_actorStartMovingTimeoutArray[_currentActorStartMovingTimeoutIndex].ActorStartMovingTimeout.register(stEventEntity, timerTime, conformation, waitHWConformation);
_actorStartMovingTimeoutArray[_currentActorStartMovingTimeoutIndex].actorID := actorID;
_actorStartMovingTimeoutArray[_currentActorStartMovingTimeoutIndex].actorPtr := actorPtr;
_actorStartMovingTimeoutArray[_currentActorStartMovingTimeoutIndex].expectedActorValue := expectedActorValue;
_actorStartMovingTimeoutArray[_currentActorStartMovingTimeoutIndex].sensorID := sensorID;
_actorStartMovingTimeoutArray[_currentActorStartMovingTimeoutIndex].sensorPtr := sensorPtr;

register := TRUE;
RETURN;
END_METHOD

// resets all ActorStartMovingTimeouts
METHOD resetAll : BOOL
VAR_INPUT
END_VAR

VAR
	i : UINT;
END_VAR
// reset all alarms
FOR i := 0 TO _currentActorStartMovingTimeoutIndex DO
	_actorStartMovingTimeoutArray[i].ActorStartMovingTimeout.reset();
END_FOR

resetAll := TRUE;
RETURN;
END_METHOD

METHOD PRIVATE resolveWatchdogInput : BOOL
VAR_INPUT
	ActorStartMovingTimeoutEx : ActorStartMovingtimeoutEx_t;
END_VAR

VAR
	_tmpStr : STRING;
	
	_sensorVal : BOOL := FALSE; 
	_actorVal : BOOL := FALSE;
END_VAR
IF _IOExpantionHandler = NULL AND _IOExpantionHandlerNotValidErrorSent = FALSE THEN
	_IOExpantionHandlerNotValidErrorSent := TRUE;
	_ErrorMessage.CreateEx(TC_EVENTS.ProgrammingErrors.NoValidPointerToIOExpantionHandler, 0 );
	_ErrorMessage.ipArguments.AddString(__POUNAME());
	_tmpStr := formatPosition(__POSITION());
	_ErrorMessage.ipArguments.AddString(_tmpStr);
	_ErrorMessage.Send(0);
	resolveWatchdogInput := FALSE;
	RETURN;
END_IF

// reslove sensor value
IF ActorStartMovingTimeoutEx.sensorPtr <> NULL THEN
	_sensorVal := ActorStartMovingTimeoutEx.sensorPtr^;
ELSIF ActorStartMovingTimeoutEx.sensorID <> sensorID_t.SENSOR_NO_SENSOR THEN
	_sensorVal := _IOExpantionHandler^.getSensorStatus(ActorStartMovingTimeoutEx.sensorID);
END_IF

// reslove actor value
IF ActorStartMovingTimeoutEx.actorPtr <> NULL THEN
	_actorVal := ActorStartMovingTimeoutEx.actorPtr^;
ELSIF ActorStartMovingTimeoutEx.actorID <> actorID_t.ACTOR_NO_ACTOR THEN
	_actorVal := _IOExpantionHandler^.getActor(ActorStartMovingTimeoutEx.actorID);
END_IF

IF _sensorVal = FALSE THEN // ignore cases when sensor isn't active
	resolveWatchdogInput := TRUE; 
	RETURN; 
END_IF

IF ActorStartMovingTimeoutEx.expectedActorValue <> _actorVal THEN
	resolveWatchdogInput := FALSE; // value missmatch, start timeout
	RETURN;
END_IF

resolveWatchdogInput := TRUE; 
RETURN;
END_METHOD

// sets the IOExpantionHandler refferance
METHOD setIOExpantionHandler : BOOL
VAR_INPUT
	IOExpantionHandlerPtr: POINTER TO IOExpantionHandler_t;
END_VAR
_IOExpantionHandler := IOExpantionHandlerPtr;
setIOExpantionHandler := TRUE;
RETURN;
END_METHOD

METHOD update : BOOL
VAR_INPUT
END_VAR

VAR
	i : UINT;
END_VAR
FOR i := 0 TO _currentActorStartMovingTimeoutIndex DO
	_actorStartMovingTimeoutArray[i].ActorStartMovingTimeout.update(resolveWatchdogInput(_actorStartMovingTimeoutArray[i]));
END_FOR

update := TRUE;
RETURN;
END_METHOD

END_FUNCTION_BLOCK

// ---- POUs/ErrorSystem/PrimitiveWatchdogManager_t.TcPOU
FUNCTION_BLOCK PrimitiveWatchdogManager_t
VAR_INPUT
END_VAR
VAR_OUTPUT
END_VAR
VAR
	_primitiveWatchdogArray : ARRAY [0..99] OF  PrimitiveWatchdogEx_t;
	_maxPrimitiveWatchdogIndex : UINT := 99;
	_currentPrimitiveWatchdogIndex : UINT := 0;
	_ErrorMessage : FB_TcMessage;
	_IOExpantionHandler : POINTER TO IOExpantionHandler_t := NULL;
	
	_IOExpantionHandlerNotValidErrorSent : BOOL := FALSE;
END_VAR

// clears and destroyes all PrimetiveWatchdogs
METHOD clear : BOOL
VAR_INPUT
END_VAR
_currentPrimitiveWatchdogIndex := 0;

clear := TRUE;
RETURN;
END_METHOD

// confirm all primitiveWatchdogs
METHOD confirmAll : BOOL
VAR_INPUT
END_VAR

VAR
	i: UINT;
END_VAR
// confirm all alarms
FOR i := 0 TO _currentPrimitiveWatchdogIndex DO
	_primitiveWatchdogArray[i].primitiveWatchdog.confirm();
END_FOR

confirmAll := TRUE;
RETURN;
END_METHOD

// if true an error has been trown
METHOD hasError : BOOL
VAR_INPUT
END_VAR

VAR
	i: UINT;
END_VAR
FOR i := 0 TO _currentPrimitiveWatchdogIndex DO
	hasError := hasError OR THIS^._primitiveWatchdogArray[i].primitiveWatchdog.isAlarmRaised();
END_FOR

RETURN;
END_METHOD

METHOD register : BOOL
VAR_INPUT
	stEventEntity : TcEventEntry;
	timerTime : TIME; // sets the timer for the timeout
	conformation : BOOL := TRUE;
	invert : BOOL := FALSE; // if true, inverts the watchdog feeding signal
	sensorID : sensorID_t := sensorID_t.SENSOR_NO_SENSOR;
	sensorPtr : POINTER TO BOOL := NULL;
	waitHWConformation : BOOL := TRUE;
END_VAR
VAR
	_tmpStr : STRING;
END_VAR
IF _currentPrimitiveWatchdogIndex + 1 > _maxPrimitiveWatchdogIndex THEN
	_ErrorMessage.CreateEx(TC_EVENTS.ProgrammingErrors.ExceedingAllowedAmountOfPrimitiveWatchdogTimeouts, 0 );
	_ErrorMessage.ipArguments.AddString(__POUNAME());
	_tmpStr := formatPosition(__POSITION());
	_ErrorMessage.ipArguments.AddString(_tmpStr);
	_ErrorMessage.ipArguments.AddUInt(_maxPrimitiveWatchdogIndex);
	_ErrorMessage.Send(0);
	
	register := FALSE;
	RETURN;
END_IF

IF (NOT(sensorID = sensorID_t.SENSOR_NO_SENSOR XOR sensorPtr = NULL)) THEN
	_ErrorMessage.CreateEx(TC_EVENTS.ProgrammingErrors.primitiveWatchdogNoValidSensorGiven, 0 );
	_ErrorMessage.ipArguments.AddString(__POUNAME());
	_tmpStr := formatPosition(__POSITION());
	_ErrorMessage.ipArguments.AddString(_tmpStr);
	_ErrorMessage.Send(0);
	
	register := FALSE;
	RETURN;
END_IF

_currentPrimitiveWatchdogIndex := _currentPrimitiveWatchdogIndex + 1; // increase it by one

_primitiveWatchdogArray[_currentPrimitiveWatchdogIndex].primitiveWatchdog.register(stEventEntity, timerTime, conformation, waitHWConformation);

_primitiveWatchdogArray[_currentPrimitiveWatchdogIndex].sensorID := sensorID;
_primitiveWatchdogArray[_currentPrimitiveWatchdogIndex].sensorPtr := sensorPtr;
_primitiveWatchdogArray[_currentPrimitiveWatchdogIndex].invert := invert;

register := TRUE;
RETURN;
END_METHOD

// resets all primitiveTimeouts
METHOD resetAll : BOOL
VAR_INPUT
END_VAR

VAR
	i: UINT;
END_VAR
// reset all alarms
FOR i := 0 TO _currentPrimitiveWatchdogIndex DO
	_primitiveWatchdogArray[i].primitiveWatchdog.reset();
END_FOR

resetAll := TRUE;
RETURN;
END_METHOD

METHOD PRIVATE resolveWatchdogImput : BOOL
VAR_INPUT
	PrimitiveWatchdogEx : PrimitiveWatchdogEx_t;
END_VAR

IF PrimitiveWatchdogEx.sensorID <> sensorID_t.SENSOR_NO_SENSOR THEN
	resolveWatchdogImput := _IOExpantionHandler^.getSensorStatus(PrimitiveWatchdogEx.sensorID);
END_IF

IF PrimitiveWatchdogEx.sensorPtr <> NULL THEN
	resolveWatchdogImput := PrimitiveWatchdogEx.sensorPtr^;
END_IF

IF PrimitiveWatchdogEx.invert THEN
	resolveWatchdogImput := NOT resolveWatchdogImput;
END_IF

RETURN;
END_METHOD

METHOD setIOExpantionHandler : BOOL
VAR_INPUT
	IOExpantionHandlerPtr: POINTER TO IOExpantionHandler_t;
END_VAR
_IOExpantionHandler := IOExpantionHandlerPtr;
setIOExpantionHandler := TRUE;
RETURN;
END_METHOD

METHOD update : BOOL
VAR_INPUT
END_VAR

VAR
	i: UINT;
END_VAR
FOR i := 0 TO _currentPrimitiveWatchdogIndex DO
	_primitiveWatchdogArray[i].primitiveWatchdog.update(resolveWatchdogImput(_primitiveWatchdogArray[i]));
END_FOR

update := TRUE;
RETURN;
END_METHOD

END_FUNCTION_BLOCK

// ---- POUs/ErrorSystem/IOExpantionMessageErrorHandler_t.TcPOU
// handles errors that can be attached from IOExpantionHandler
FUNCTION_BLOCK IOExpantionMessageErrorHandler_t
VAR_INPUT
END_VAR
VAR_OUTPUT
END_VAR
VAR
	_IOExpantionMessageErrorArray : ARRAY [0..99] OF  IOExpantionMessageErrorEx_t;
	_maxIOExpantionMessageErrorIndex : UINT := 99;
	_currentIOExpantionMessageErrorIndex : UINT := 0;
	_ErrorMessage : FB_TcMessage;
	_IOExpantionHandler : POINTER TO IOExpantionHandler_t := NULL;
	
	_IOExpantionHandlerNotValidErrorSent : BOOL := FALSE;
	
	_PrimitiveWatchdogManager : PrimitiveWatchdogManager_t;
END_VAR

// clears and deletes all IOExpantionMessageErrors
METHOD clear : BOOL
VAR_INPUT
END_VAR
VAR
	i : uint := 0;
END_VAR
_PrimitiveWatchdogManager.clear();

FOR i := 0 TO _currentIOExpantionMessageErrorIndex DO 
	_IOExpantionHandler^.unsubscribe(ADR(_IOExpantionMessageErrorArray[i].clearMessageCallback));
	_IOExpantionHandler^.unsubscribe(ADR(_IOExpantionMessageErrorArray[i].errorMessageCallback));
END_FOR

_currentIOExpantionMessageErrorIndex := 0;

clear := TRUE;
return;
END_METHOD

// confirm all errors
METHOD confirmAll : BOOL
VAR_INPUT
END_VAR
VAR
	i : UINT := 0;
END_VAR
confirmAll := _PrimitiveWatchdogManager.confirmAll();
return;
END_METHOD

// if true an error has been trown
METHOD hasError : BOOL
VAR_INPUT
END_VAR
hasError := _PrimitiveWatchdogManager.hasError();
return;
END_METHOD

// registers a new error
METHOD register : BOOL
VAR_INPUT
	stEventEntity : TcEventEntry;
	timerTime : TIME; // sets the timer for the timeout
	conformation : BOOL := TRUE;
	diagCodeErrorMessage : ARRAY[0..3] OF BYTE;
	textIDErrorMessage : ARRAY [0..1] OF BYTE;
	diagCodeClearMessage : ARRAY[0..3] OF BYTE;
	textIDClearMessage : ARRAY [0..1] OF BYTE;
END_VAR
_currentIOExpantionMessageErrorIndex := _currentIOExpantionMessageErrorIndex + 1; // increase it by one


//_IOExpantionMessageErrorArray[_currentIOExpantionMessageErrorIndex]
_IOExpantionHandler^.subscribe(callbackVariable := ADR(_IOExpantionMessageErrorArray[_currentIOExpantionMessageErrorIndex].errorMessageCallback), diagCode := diagCodeErrorMessage, textID := textIDErrorMessage);
_IOExpantionHandler^.subscribe(callbackVariable := ADR(_IOExpantionMessageErrorArray[_currentIOExpantionMessageErrorIndex].clearMessageCallback), diagCode := diagCodeClearMessage, textID := textIDClearMessage);

_PrimitiveWatchdogManager.register(stEventEntity := stEventEntity, timerTime := timerTime, conformation := conformation, invert := true, sensorPtr := ADR(_IOExpantionMessageErrorArray[_currentIOExpantionMessageErrorIndex].isErrorActive), waitHWConformation := TRUE);

register := TRUE;
return;
END_METHOD

METHOD resetAll : BOOL
VAR_INPUT
END_VAR
resetAll := _PrimitiveWatchdogManager.resetAll();
return;
END_METHOD

// this method directly changes the IOExpantionMessageErrorEx_t
METHOD PRIVATE resolveWatchdogInput : BOOL
VAR_INPUT
	IOExpantionMessageErrorEx : REFERENCE TO IOExpantionMessageErrorEx_t;
END_VAR

IOExpantionMessageErrorEx.isErrorActive := IOExpantionMessageErrorEx.isErrorActive OR IOExpantionMessageErrorEx.errorMessageCallback;
IOExpantionMessageErrorEx.errorMessageCallback := FALSE;


IOExpantionMessageErrorEx.isErrorActive := IOExpantionMessageErrorEx.isErrorActive AND (NOT IOExpantionMessageErrorEx.clearMessageCallback);
IOExpantionMessageErrorEx.clearMessageCallback := FALSE;

resolveWatchdogInput := IOExpantionMessageErrorEx.isErrorActive;
RETURN;
END_METHOD

METHOD setIOExpantionHandler : BOOL
VAR_INPUT
	IOExpantionHandlerPtr : POINTER TO IOExpantionHandler_t;
END_VAR
_IOExpantionHandler := IOExpantionHandlerPtr;
_PrimitiveWatchdogManager.setIOExpantionHandler(_IOExpantionHandler);
setIOExpantionHandler := TRUE;
RETURN;
END_METHOD

METHOD update : BOOL
VAR_INPUT
END_VAR
VAR
	i : UINT := 0;
END_VAR
_PrimitiveWatchdogManager.update();

FOR i := 0 TO _currentIOExpantionMessageErrorIndex DO
	resolveWatchdogInput(_IOExpantionMessageErrorArray[i]);
END_FOR

update := TRUE;
RETURN;
END_METHOD

END_FUNCTION_BLOCK

// ---- POUs/ARCommunication/ARDeviceErrorSystemLinker_t.TcPOU
// this class may be used to translate alarms from the EventLogger to a bool value and attach this to the ARDeviceAPI_t
FUNCTION_BLOCK ARDeviceErrorSystemLinker_t
VAR_INPUT
END_VAR
VAR_OUTPUT
END_VAR
VAR
	_EventLogger : FB_TcEventLogger;
	_ErrorMessage : FB_TcMessage;
	
	_linksArray : ARRAY[0..99] OF ARDeviceErrorSystemLink_t;
	_currentLinksArrayIndex : UINT := 0;
	_maxLinksArrayIndex : UINT := 99;
END_VAR

// clears all registered links
METHOD clear : BOOL
VAR_INPUT
END_VAR
VAR
	i : UINT := 0;
END_VAR
FOR i := 0 TO _maxLinksArrayIndex DO
	_linksArray[i].callBackPtr := NULL;
END_FOR

_currentLinksArrayIndex := 0;
clear := TRUE;
return;
END_METHOD

// register a link
METHOD register : BOOL
VAR_INPUT
	stEventEntity : TcEventEntry; 
	callBackPtr : POINTER TO BOOL; // pointer to variable from ARDeviceAPI_t
END_VAR

VAR
	_tmpStr : STRING;
END_VAR
IF _currentLinksArrayIndex + 1 > _maxLinksArrayIndex THEN
	_ErrorMessage.CreateEx(TC_EVENTS.ProgrammingErrors.ExceedingAllowedAmountOfLinks, 0 );
	_ErrorMessage.ipArguments.AddString(__POUNAME());
	_tmpStr := formatPosition(__POSITION());
	_ErrorMessage.ipArguments.AddString(_tmpStr); 
	_ErrorMessage.ipArguments.AddUInt(_maxLinksArrayIndex);
	_ErrorMessage.Send(0);
	
	register := FALSE;
	RETURN;
END_IF

_currentLinksArrayIndex := _currentLinksArrayIndex + 1;

_linksArray[_currentLinksArrayIndex].callBackPtr := callBackPtr;
_linksArray[_currentLinksArrayIndex].stEventEntity := stEventEntity;

register := TRUE;
return;
END_METHOD

// call this every cycle
METHOD update : BOOL
VAR_INPUT
END_VAR

VAR
	i : UINT;
	_alarm : FB_TcAlarm;
END_VAR
FOR i := 1 TO _maxLinksArrayIndex DO
	IF _linksArray[i].callBackPtr <> NULL THEN
		_EventLogger.GetAlarmEx(stEventEntry := _linksArray[i].stEventEntity,fbAlarm := _alarm);
		_linksArray[i].callBackPtr^ := _alarm.bActive;
	END_IF
END_FOR

update := TRUE;
return;
END_METHOD

END_FUNCTION_BLOCK

// ---- POUs/ARCommunication/ARDeviceErrorSystemLinkerInitialiser.TcPOU
// links and initialises the ARDeviceErrorSystemLinker_t to the ARDeviceAPI_t. Call tis functon only at startup and once
FUNCTION ARDeviceErrorSystemLinkerInitialiser : BOOL
VAR_INPUT
	ARDeviceSystemLinker : REFERENCE TO ARDeviceErrorSystemLinker_t;
	ARDeviceAPI : Reference to ARDeviceAPI_t;
END_VAR
VAR
END_VAR


ARDeviceSystemLinker.register(stEventEntity := TC_EVENTS.OperationalErrors2.LowPneumaticPressure, ADR(ErrorSystemStatusVar.errorHide_ERR_PNEU_LOW_PR_402));
ARDeviceSystemLinker.register(stEventEntity := TC_EVENTS.OperationalErrors2.LinearDriveStartMoveLeftTimeout, ADR(ErrorSystemStatusVar.errorHide_ERR_LD_START_LEFT_408_TIMEOUT));
ARDeviceSystemLinker.register(stEventEntity := TC_EVENTS.OperationalErrors2.LinearDriveStartMoveRightTimeout, ADR(ErrorSystemStatusVar.errorHide_ERR_LD_START_RIGHT_408_TIMEOUT));
ARDeviceSystemLinker.register(stEventEntity := TC_EVENTS.OperationalErrors2.LinearDriveMoveTimedout, ADR(ErrorSystemStatusVar.errorHide_ERR_LD_MOVE_408_TIMEOUT));
ARDeviceSystemLinker.register(stEventEntity := TC_EVENTS.OperationalErrors2.RotaryTableMoveTimeout, ADR(ErrorSystemStatusVar.errorHide_ERR_RT_MOVE_408_TIMEOUT));
ARDeviceSystemLinker.register(stEventEntity := TC_EVENTS.OperationalErrors2.Y2moveTimeout, ADR(ErrorSystemStatusVar.errorHide_ERR_Y2_MOVE_408_TIMEOUT));
ARDeviceSystemLinker.register(stEventEntity := TC_EVENTS.OperationalErrors2.Y2StartMoveDownTimeout, ADR(ErrorSystemStatusVar.errorHide_ERR_Y2_START_DOWN_408_TIMEOUT));
ARDeviceSystemLinker.register(stEventEntity := TC_EVENTS.OperationalErrors2.Y2StartMoveUpTimeout, ADR(ErrorSystemStatusVar.errorHide_ERR_Y2_START_UP_408_TIMEOUT));
ARDeviceSystemLinker.register(stEventEntity := TC_EVENTS.OperationalErrors2.Y3moveTimeout, ADR(ErrorSystemStatusVar.errorHide_ERR_Y3_MOVE_408_TIMEOUT));
ARDeviceSystemLinker.register(stEventEntity := TC_EVENTS.OperationalErrors2.Y3StartMoveDownTimeout, ADR(ErrorSystemStatusVar.errorHide_ERR_Y3_START_DOWN_408_TIMEOUT));
ARDeviceSystemLinker.register(stEventEntity := TC_EVENTS.OperationalErrors2.Y3StartMoveUpTimeout, ADR(ErrorSystemStatusVar.errorHide_ERR_Y3_START_UP_408_TIMEOUT));

ARDeviceErrorSystemLinkerInitialiser := true;
RETURN;

END_FUNCTION

// ---- POUs/ARCommunication/Websocket/ARCommunicationWSExtentionWS_t.TcPOU
{attribute 'c++_compatible'}
// class for implementing IotWebSocetClient functions without exposing them may only be used for ARCommunication_t
FUNCTION_BLOCK ARCommunicationWSExtentionWS_t EXTENDS FB_IotWebSocketClient
VAR_INPUT
END_VAR
VAR_OUTPUT
	lastMessage : STRING(255) := ''; // last recived message
END_VAR
VAR	
	_newMessageAvalable : BOOL := FALSE; // is set true whenever a new message arrives
END_VAR

PROPERTY newMessageAvalable : bool
GET
newMessageAvalable :=  _newMessageAvalable;
END_GET
SET
_newMessageAvalable := newMessageAvalable;
END_SET
END_PROPERTY

{attribute 'TcTypeSystem'}
{attribute 'c++_compatible'}
{attribute 'minimal_input_size' := '4'}
{attribute 'pack_mode' := '4'}
{attribute 'TcRpcEnable'}
METHOD OnWebSocketClose : Global.HRESULT
VAR_INPUT
	statusCode	: UINT;
	content	: Global.PVOID;
	contentLength	: UDINT;
END_VAR
END_METHOD

{attribute 'TcTypeSystem'}
{attribute 'c++_compatible'}
{attribute 'minimal_input_size' := '4'}
{attribute 'pack_mode' := '4'}
{attribute 'TcRpcEnable'}
METHOD OnWebSocketMessage : Global.HRESULT
VAR_INPUT
	content	: Global.PVOID;
	contentLength	: UDINT;
	contentType	: Global.ETcIotWebSocketContentType;
END_VAR
VAR
	ptr : POINTER TO STRING;
END_VAR
// if it isn't text, drop packet
IF  contentType = Global.ETcIotWebSocketContentType.WS_CONTENT_TEXT THEN
		ptr := content;
		THIS^.lastMessage := ptr^;
		THIS^._newMessageAvalable := TRUE;	
END_IF
END_METHOD

{attribute 'TcTypeSystem'}
{attribute 'c++_compatible'}
{attribute 'minimal_input_size' := '4'}
{attribute 'pack_mode' := '4'}
{attribute 'TcRpcEnable'}
METHOD OnWebSocketOpen : Global.HRESULT
VAR_IN_OUT CONSTANT
	webSocketProtocol	: STRING;
	origin	: STRING;
END_VAR
VAR_INPUT
	bPerMessageDeflate	: BOOL;
END_VAR
END_METHOD

{attribute 'TcTypeSystem'}
{attribute 'c++_compatible'}
{attribute 'minimal_input_size' := '4'}
{attribute 'pack_mode' := '4'}
METHOD TcAddRef : UDINT
END_METHOD

{attribute 'TcTypeSystem'}
{attribute 'c++_compatible'}
{attribute 'minimal_input_size' := '4'}
{attribute 'pack_mode' := '4'}
METHOD TcQueryInterface : Global.HRESULT
VAR_INPUT
	iid	: REFERENCE TO Global.IID;
	pipItf	: POINTER TO Global.PVOID;
END_VAR
END_METHOD

{attribute 'TcTypeSystem'}
{attribute 'c++_compatible'}
{attribute 'minimal_input_size' := '4'}
{attribute 'pack_mode' := '4'}
METHOD TcRelease : UDINT
END_METHOD

END_FUNCTION_BLOCK

// ---- POUs/ARCommunication/Websocket/ARCommunicationWS_t.TcPOU
// abstracts the ARCommunicationWSExtention
FUNCTION_BLOCK ARCommunicationWS_t 
VAR_INPUT
END_VAR
VAR_OUTPUT
END_VAR
VAR
	_ARDevice : ARCommunicationWSExtentionWS_t;
	_initialConnect : BOOL := FALSE;
END_VAR

METHOD getConnectionStatus : BOOL
VAR_INPUT
END_VAR
// gets the communication status of the connection
getConnectionStatus := _ARDevice.bConnected;
return;
END_METHOD

// gets the last saved message from the client (max str length 255)
METHOD getLastMessage : STRING(255)
VAR_INPUT
END_VAR
getLastMessage := _ARDevice.lastMessage;

_ARDevice.newMessageAvalable := FALSE;
END_METHOD

METHOD newMessageRecived : BOOL
VAR_INPUT
END_VAR
// returns if a new message has been recived
newMessageRecived := _ARDevice._newMessageAvalable;
END_METHOD

METHOD sendNewMessage : BOOL
VAR_INPUT
	str : STRING(255); // (max str length 255)
END_VAR
// sends a new message to the client
_ARDevice.SendMessage(pContent := ADR(str), nContentSize := SIZEOF(str), bTextContent := TRUE, bCompress := FALSE);
END_METHOD

METHOD PRIVATE startConnection : BOOL
VAR_INPUT
END_VAR
IF _ARDevice.bConnected THEN
	RETURN;
END_IF


_ARDevice.nHostPort := 1880;
_ARDevice.sHostName := 'localhost';
_ARDevice.sUri := 'ws/PLC';
_ARDevice.bKeepAlive := FALSE;
_ARDevice.nConnectResponseTimeout := 60;
_ARDevice.nKeepAliveCloseTimeout := 60;
//_ARDevice.stTLS.bNoServerCertCheck := TRUE;
_ARDevice.bPerMessageDeflate := FALSE;
_ARDevice.sOrigin := 'ws/PLC';
_ARDevice.Connect(TRUE);
END_METHOD

METHOD PRIVATE stopConnection : BOOL
VAR_INPUT
END_VAR
IF NOT _ARDevice.bConnected THEN
	RETURN;
END_IF

_ARDevice.Disconnect();
END_METHOD

// is called every cycle, used to upholed communication and check if a new message has been recived
METHOD update : BOOL
VAR_INPUT
END_VAR
IF _initialConnect = FALSE THEN // initial connection
	_initialConnect := true;
	THIS^.startConnection();
END_IF

IF _ARDevice.eConnectionState = ETcIotWebSocketStatus.WS_STATUS_SOCK_NO_CONN THEN 
	//THIS^.stopConnection();
END_IF

IF _ARDevice.bConnected = FALSE AND _ARDevice.eConnectionState <> ETcIotWebSocketStatus.WS_STATUS_BUSY THEN // retry if connection is lost
	//THIS^.startConnection();
END_IF

_ARDevice.Execute();
END_METHOD

END_FUNCTION_BLOCK

// ---- POUs/ErrorSystem/GernericErrorWatchdog_t.TcPOU
FUNCTION_BLOCK GernericErrorWatchdog_t  
VAR_INPUT
END_VAR
VAR_OUTPUT
END_VAR
VAR
	_alarm : FB_TcAlarm; 	// the alarm object
	_init : BOOL := FALSE;  // if true the object is initialised
	_timer : TON; 			// counts the time
	_sensor : BOOL; 		// if true reset timer
	_isAlarmDisplayed : BOOL := FALSE; // if true, the alarm wasn't deleted from the event logger 
	_isAlarmClearedLast : BOOL := FALSE; // true when the alarm has been cleard last
	_waitHWConformation : BOOL := TRUE; // if true, the watchdogs wait for the correct value bevore clearing the error.
	
	_eventLogger : FB_TcEventLogger;
	_eventLoggerSettings : FB_TcClearLoggedEventsSettings;
	_eventLoggerFilter : FB_TcEventFilter;
END_VAR

// confirm the alarm
METHOD confirm : BOOL
VAR_INPUT
END_VAR
IF _init = FALSE THEN
	confirm := FALSE; 
	RETURN;
END_IF

_alarm.Confirm();

// restet timeout
_timer.IN := FALSE;
_timer();

confirm := TRUE;
END_METHOD

// returns true if the alarm is raised
METHOD isAlarmRaised : BOOL
VAR_INPUT
END_VAR
IF _init = FALSE THEN
	isAlarmRaised := FALSE;
	return;
END_IF

isAlarmRaised := _alarm.bActive;
RETURN;
END_METHOD

// registers a error state or reregister an existing error state
METHOD register : bool
VAR_INPUT
	stEventEntity : TcEventEntry;
	timerTime : TIME; // sets the timer for the timeout
	conformation : BOOL := TRUE; 
	waitHWConformation : bool := TRUE;
END_VAR
_alarm.CreateEx(stEventEntity, conformation);
_timer.PT := timerTime;
_init := TRUE;
_waitHWConformation := waitHWConformation; 
RETURN;
END_METHOD

// resets the alarm. Only use this as a last resort.
METHOD reset : BOOL
VAR_INPUT
END_VAR
IF _init = FALSE THEN
	reset := FALSE;
	RETURN;
END_IF

_alarm.Confirm();
_alarm.Clear(bResetConfirmation := TRUE);

_timer.IN := FALSE;
_timer(); 

reset := TRUE;
RETURN;
END_METHOD

// call this function every cycle. 
METHOD update : bool
VAR_INPUT
	sensor : bool; // if true the sensor is active and the watchdog resets, if it isn't set, the time starts.
END_VAR
IF _init = FALSE THEN
	update := FALSE; 
	RETURN;
END_IF



IF sensor = FALSE THEN
	_timer.IN := TRUE;
ELSE 
	_timer.IN := FALSE;
END_IF

_timer();

// clear alarm from log
IF (_alarm.bActive = FALSE AND _isAlarmDisplayed) OR _isAlarmClearedLast THEN
	_isAlarmDisplayed := FALSE;
	_isAlarmClearedLast := FALSE;
	_eventLoggerFilter.EventClass.EqualTo(value := _alarm.EventClass);
	_eventLoggerSettings.AddFilter(_eventLoggerFilter);
	_eventLogger.ClearLoggedEvents(_eventLoggerSettings);
	_eventLogger.ClearLoggedEvents(_eventLoggerSettings);
END_IF

IF _timer.Q AND _alarm.bActive = FALSE THEN
	// timeout detected
	_alarm.Raise(); 
	_isAlarmDisplayed := TRUE; 
END_IF

IF _alarm.bRaised AND (sensor OR _waitHWConformation = FALSE) THEN
	_alarm.Clear();
	_isAlarmClearedLast := NOT _alarm.bActive;
END_IF

update := TRUE;
RETURN;
END_METHOD

END_FUNCTION_BLOCK

// ---- POUs/ErrorSystem/SendErrorMessage.TcPOU
FUNCTION SendErrorMessage : BOOL
VAR_INPUT
	message : REFERENCE TO FB_TcMessage;
	position : STRING;
	POUNAME : STRING;
END_VAR
VAR
	_tmpStr : STRING;
END_VAR

message.ipArguments.AddString(__POUNAME());
_tmpStr := formatPosition(__POSITION());
message.ipArguments.AddString(_tmpStr);
message.Send(0);

SendErrorMessage := TRUE;
RETURN;

END_FUNCTION
